# EPICS substitutions: db/Beckhoff_MX/ecmcMS1110-0000.substitutions
#- MS1110-0000 is a passive EtherCAT extension and exposes no process data.
file "empty.template" {
  pattern {}
}
